(* CODESYS project bf.project

Project tree, tasks and I/O mapping:
  Device : CODESYS Control Win V3, 3S - Smart Software Solutions GmbH, order no. 305021, version 3.5.11.30
    application Application
      libraries: Standard, * (System)
      task MainTask (cyclic, interval t#20ms, priority 1) calls PLC_PRG
      program PLC_PRG [ST]
      function block MyFB [ST]
      data type ModeBlk
      data type ds33
*)

// Device/Application/ModeBlk
{attribute 'qualified_only'}
{attribute 'strict'}
TYPE ModeBlk :
(
	OutOfService := 0,
	Manual,
	Auto,
	Cas
);
END_TYPE

// Device/Application/ds33
TYPE ds33 :
STRUCT
	Value: REAL;
	Status: BOOL;
END_STRUCT
END_TYPE

// Device/Application/PLC_PRG
PROGRAM PLC_PRG
VAR
	FB1:MyFB;
	FB2:MyFB;
	in1:ds33;
	in2:ds33;
	out1:ds33;
END_VAR

FB1(in:={10,1}, casin:={20,1}, out => out1);

END_PROGRAM

// Device/Application/MyFB
FUNCTION_BLOCK MyFB
VAR_INPUT
	in: ds33;
	casin: ds33;
END_VAR

VAR_OUTPUT
	out: ds33;
END_VAR

VAR
	Mode: ModeBlk;
	sp: REAL :=5.0;
	gain:REAL := 2.0;
	auxValue: REAL;
END_VAR

out.Status := in.Status AND casin.Status;

IF (out.Status = TRUE) THEN 
	CASE Mode OF
		Modeblk.Auto :
			out.Value := (in.Value - sp)*gain;
		Modeblk.Cas :
			out.Value:=(in.Value-casin.Value)*gain;
		Modeblk.Manual:
			out.Value:=auxValue;
	END_CASE
ELSE
	out.Value := 255;
END_IF

END_FUNCTION_BLOCK
